INTERFACE ITF_Can_Supply EXTENDS ITF_PackML

{warning 'add method implementation '}
METHOD Abort : BOOL
END_METHOD

{warning 'add method implementation '}
METHOD Aborting_SC : BOOL
END_METHOD

{warning 'add method implementation '}
METHOD Auto : BOOL
END_METHOD

{warning 'add method implementation '}
METHOD Clear : BOOL
END_METHOD

{warning 'add method implementation '}
METHOD Clearing_SC : BOOL
END_METHOD

{warning 'add method implementation '}
METHOD Completing_SC : BOOL
END_METHOD

{warning 'add method implementation '}
METHOD Execute_SC : BOOL
END_METHOD

{warning 'add method implementation '}
METHOD FB_init : BOOL
VAR_INPUT
	bInitRetains : BOOL; // if TRUE, the retain variables are initialized (warm start / cold start)
	bInCopyCode : BOOL;  // if TRUE, the instance afterwards gets moved into the copy code (online change)
END_VAR
END_METHOD

{warning 'add method implementation '}
METHOD Hold : BOOL
END_METHOD

{warning 'add method implementation '}
METHOD Holding_SC : BOOL
END_METHOD

{warning 'add method implementation '}
METHOD Manueel : BOOL
END_METHOD

{warning 'add method implementation '}
METHOD Reset : BOOL
END_METHOD

{warning 'add method implementation '}
METHOD Resetting_SC : BOOL
END_METHOD

{warning 'add method implementation '}
METHOD Start : BOOL
END_METHOD

{warning 'add method implementation '}
METHOD Starting_SC : BOOL
END_METHOD

{warning 'add property implementation'}
PROPERTY State : E_State_PackML
GET
END_GET
END_PROPERTY

{warning 'add method implementation '}
METHOD Stop : BOOL
END_METHOD

{warning 'add method implementation '}
METHOD Stopping_SC : BOOL
END_METHOD

{warning 'add method implementation '}
METHOD Suspend : BOOL
END_METHOD

{warning 'add method implementation '}
METHOD Suspending_SC : BOOL
END_METHOD

{warning 'add method implementation '}
METHOD Unhold : BOOL
END_METHOD

{warning 'add method implementation '}
METHOD Unholding_SC : BOOL
END_METHOD

{warning 'add method implementation '}
METHOD Unsuspend : BOOL
END_METHOD

{warning 'add method implementation '}
METHOD Unsuspending_SC : BOOL
END_METHOD

{warning 'add method implementation '}
METHOD ZeroAllVar : BOOL
END_METHOD

END_INTERFACE

(* stored: Version 1.1.0.1, ProductVersion 3.1.4024.12
   Itf ITF_Can_Supply: Id {be7d18ee-7936-4035-920e-6c9d83390de9}
   Folder Methods: Id {9825e394-832a-471d-bf1c-71980f25670b}
   Folder Properties: Id {61811a0d-6ae7-4dd3-838e-6564c22290dc}
   Method Abort: Id {f3036df1-a8b7-4e01-8435-d3694475b554}
   Method Aborting_SC: Id {dede9959-06e9-4ae6-92d5-f759fa6a0711}
   Method Auto: Id {973a3595-3042-468b-b69d-22767af63f3a}
   Method Clear: Id {7a38a923-482d-4861-9315-89cfe0c296de}
   Method Clearing_SC: Id {786080b1-c259-417f-9800-c12d15c0e8a8}
   Method Completing_SC: Id {dfeeae52-456c-46cc-8732-d2f7c6f2a4ec}
   Method Execute_SC: Id {465dfd5c-7180-47db-aa8a-ac01e08d744e}
   Method FB_init: Id {c740385f-9f70-4a43-b200-37cf9abee838}
   Method Hold: Id {ea24847d-59eb-43cc-bec6-43dcf6f55682}
   Method Holding_SC: Id {75d0e30c-416f-41a6-8be3-d368589ec93c}
   Method Manueel: Id {99c37bf6-e5c1-48cd-9d07-8b842bf9c3c0}
   Method Reset: Id {c4a0a244-05b7-40f7-a199-9634c2056ae8}
   Method Resetting_SC: Id {bb872d1a-3ff5-47ed-a2db-7e35acf1ac95}
   Method Start: Id {9183cd8f-42e2-4ba8-8515-790ac74e3089}
   Method Starting_SC: Id {2a34f45f-8f3c-4075-ae9f-b84fdc2c2dd4}
   Property State: Id {4a8a11d1-a82f-4c23-914e-479f7db93af8}
   Get Get: Id {b6e868ca-878f-4b3a-a1c8-39f62a723a8d}
   Method Stop: Id {7895009c-a899-431c-804d-815ba92f02e4}
   Method Stopping_SC: Id {704aedf8-388c-4b8c-bd30-93f42701868c}
   Method Suspend: Id {cbd13e4c-e80f-496e-b1c4-4547acc74546}
   Method Suspending_SC: Id {ee7dd256-fb6f-425a-9fb4-1c97880a63fa}
   Method Unhold: Id {808ceb9e-32ff-42ed-8798-8542f8f1cc5c}
   Method Unholding_SC: Id {85803510-1a31-4e6a-886b-0e537a5f36b6}
   Method Unsuspend: Id {136f031f-19d1-4e3f-80a4-ea1f156aa0c8}
   Method Unsuspending_SC: Id {695786f1-4de6-44e8-917a-6aa058954565}
   Method ZeroAllVar: Id {46bf6cc3-ccb7-47fe-81d9-b0a3f45a9c6c} *)
